(* IEC 61131-3 sources: Industry-PLC-LLM/data/PLCBEAD_repo/PLCBEAD_PLCEmbed-main/PLC-BEAD/Source/GEB/GEO_TO_DEG, 1 file *)

(* ---- GEO_TO_DEG.ST ---- *)
FUNCTION GEO_TO_DEG:REAL

	VAR_INPUT
		D :	INT;
		M :	INT;
		SEC :	REAL;
	END_VAR

	GEO_TO_DEG := INT_TO_REAL(D) + INT_TO_REAL(M) * 0.016666666666667 + SEC * 0.00027777777777778;

END_FUNCTION

PROGRAM program0
  VAR
    D :	INT;
	M :	INT;
	SEC :	REAL;
    LocalOUT  : REAL;
  END_VAR

  LocalOUT := GEO_TO_DEG(D, M, SEC);
END_PROGRAM
